{attribute 'linkalways'} 
{attribute 'no_explicit_call' := 'This FB is a CLASS and must be accessed using methods or properties'}
{attribute 'enable_dynamic_creation'}
FUNCTION_BLOCK Node_F_VN_MaxElementElementwise_TcVnVector3_SINT EXTENDS VisionNode
VAR
    ipContainer : _ITcVnContainer;
    aMax : _TcVnVector3_SINT;
    hrPrev : _HRESULT(S_OK);
    hresult : _HRESULT(S_OK);
END_VAR

METHOD PUBLIC  Clone : I_Node
VAR
	pNode : POINTER TO Node_F_VN_MaxElementElementwise_TcVnVector3_SINT;
END_VAR
pNode := __NEW(Node_F_VN_MaxElementElementwise_TcVnVector3_SINT);
Clone := pNode^;
END_METHOD

METHOD FB_init : BOOL
VAR_INPUT
	bInitRetains : BOOL; // if TRUE, the retain variables are initialized (warm start / cold start)
	bInCopyCode : BOOL;  // if TRUE, the instance afterwards gets moved into the copy code (online change)
END_VAR
AddInput('ipContainer', ipContainer);
AddInput('hrPrev', hrPrev);
AddOutput('ipContainer', ipContainer);
AddOutput('aMax', aMax);
AddOutput('hresult',hresult);
END_METHOD

METHOD PROTECTED OnExecute
hresult.Value := F_VN_MaxElementElementwise_TcVnVector3_SINT(
    ipContainer := ipContainer.Value,
    aMax := aMax.Value,
    hrPrev:= hrPrev.Value);
END_METHOD

METHOD PUBLIC PreExecutionCheck
VAR_INPUT
	Check : I_PreExecutionChecks;
END_VAR
Check.IsTrue(ipContainer.IsValid, 'ipContainer must be a valid container');
Check.IsTrue(ipContainer.IsType(TC_GLOBAL_CONST_LIST.ContainerType_Vector_TcVnVector3_SINT), 'ipContainer contains incorrect type');
END_METHOD

END_FUNCTION_BLOCK

(* stored: Version 1.1.0.1, ProductVersion 3.1.4026.13
   POU Node_F_VN_MaxElementElementwise_TcVnVector3_SINT: Id {a0e636ab-c68b-477a-b278-84459ab16f89}, SpecialFunc None
   Folder Constructor: Id {dc150795-d569-4fa9-a0e1-4962ac1e5537}
   Method Clone: Id {d01711bf-1fe4-4545-a6d3-d8887757e613}
   Method FB_init: Id {e1916464-43c8-4c82-8167-8faf22b09911}
   Method OnExecute: Id {2834e8e8-5f7b-48ae-8766-1f74a3573448}
   Method PreExecutionCheck: Id {dde71d66-3cae-4f16-a741-f974cbc9899c} *)
